// TIA Portal V20 export
DATA_BLOCK "DB_SafetyStandard"   // DB20
// stored: Access Published, MemoryReserve 100
   VAR
      ToStandard : Struct
         EstopActive : Bool;
      END_STRUCT;
      PressReset : Bool;
      ToHMI : Struct
         "EstopPB -AS1.7.4 -SF09 -Zone2" : Bool;
         "EstopPB -AS1.12.3 -SF10 -Zone3" : Bool;
         "EstopPB -AS1.13.14 -SF11 -Zone3" : Bool;
         "EstopPB -AS1.55.2 -SF01 -Zone1" : Bool;
         "EstopPB -AS1.55.11 -SF02 -Zone1" : Bool;
         "EstopPB -AS1.55.18 -SF03 -Zone1" : Bool;
         "EstopPB -AS1.58.2 -SF04 -Zone1" : Bool;
         "EstopPB -AS1.58.11 -SF05 -Zone1" : Bool;
         "EstopPB -AS1.58.19 -SF06 -Zone1" : Bool;
         "EstopPB -AS1.5.9 -SF07 -Zone2" : Bool;
         "EstopPB -AS1.9.4 -SF08 -Zone2" : Bool;
         "EstopPB -MCC100 -402SF7" : Bool;
         "PhaseOK -MCC100" : Bool;
         "EstopPB -AS1.50.7 -SF21" : Bool;
         "EstopPB -AS1.50.24 -SF22" : Bool;
         "EstopPB -AS1.50.8 -SF23" : Bool;
         "EstopPB -BP1.2.42 -SF24" : Bool;
         "EstopPB -BP2.3.2 -SF25" : Bool;
         "EstopPB -BP1.14.3 -SF26" : Bool;
         "EstopPB -BP1.6.2 -SF27" : Bool;
         "EstopPB -MCC300 -402SF7" : Bool;
         "PhaseOK -MCC300" : Bool;
      END_STRUCT;
      holdAlarmOffTimer : TON_TIME;
      holdAlarmOff : Bool;
   END_VAR
BEGIN
END_DATA_BLOCK
